(* IEC 61131-3 sources: repolevel_ST_code_completion/output/0122完整版本_无planner目前sota/repoeval_Decorator_Application/readful_result_history, 10 files *)

(* ---- ConcreteComponment_0.st ---- *)
{attribute 'enable_dynamic_creation'}
//This class creates the most basic object well called. This object is to be decorated
FUNCTION_BLOCK ConcreteComponent IMPLEMENTS Component_Interface
VAR_INPUT
END_VAR
VAR_OUTPUT
END_VAR
VAR
	sDescription : STRING;
	rValue : REAL;
END_VAR

METHOD CreateObject : BOOL
VAR
	tempDescription : STRING;
	tempValue : REAL;
END_VAR

tempDescription := 'Basic Object';
tempValue := 0.0;

sDescription := tempDescription;
rValue := tempValue;

CreateObject := TRUE;
RETURN;
END_FUNCTION_BLOCK

(* ---- ConcreteComponment_1.st ---- *)
{attribute 'enable_dynamic_creation'}
//This class creates the most basic object well called. This object is to be decorated
FUNCTION_BLOCK ConcreteComponent IMPLEMENTS Component_Interface
VAR_INPUT
END_VAR
VAR_OUTPUT
END_VAR
VAR
  sDescription : STRING;
  rValue : REAL;
  tempDescription : STRING; // Moved from invalid nested VAR block
  tempValue : REAL;         // Moved from invalid nested VAR block
END_VAR

// Replacing METHOD with simple implementation logic
tempDescription := 'Basic Object';
tempValue := 0.0;

sDescription := tempDescription;
rValue := tempValue;

RETURN;
END_FUNCTION_BLOCK

(* ---- ConcreteComponment_2.st ---- *)
{attribute 'enable_dynamic_creation'}
//This class creates the most basic object well called. This object is to be decorated
FUNCTION_BLOCK ConcreteComponent // Removed IMPLEMENTS Component_Interface
VAR_INPUT
END_VAR
VAR_OUTPUT
END_VAR
VAR
 sDescription : STRING;
 rValue : REAL;
 tempDescription : STRING; // Moved from invalid nested VAR block
 tempValue : REAL;         // Moved from invalid nested VAR block
END_VAR

// Replacing METHOD with simple implementation logic
tempDescription := 'Basic Object';
tempValue := 0.0;

sDescription := tempDescription;
rValue := tempValue;

RETURN;
END_FUNCTION_BLOCK

(* ---- ConcreteDecoratorA_0.st ---- *)
{attribute 'enable_dynamic_creation'}
//This class acts as a decorating class. It adds responsibilities and functionality to the component
FUNCTION_BLOCK ConcreteDecoratorA EXTENDS Decorator
VAR_INPUT
	//Reference to store the component to be decorated
	tempInputComponent : Component_Interface;
END_VAR
VAR_OUTPUT
END_VAR
VAR
	// Local variables to store additional functionality
	additionalDescription : STRING;
	additionalValue : REAL;
END_VAR

// Logic to add responsibilities and functionality to the component
tempComponent := tempInputComponent;

// Add additional description to the component
additionalDescription := ' - Decorated by ConcreteDecoratorA';
sDescription := tempComponent.GetDescription() + additionalDescription;

// Add additional value to the component
additionalValue := 10.0; // Example value to add
rValue := tempComponent.GetValue() + additionalValue;
END_FUNCTION_BLOCK

(* ---- ConcreteDecoratorB_0.st ---- *)
{attribute 'enable_dynamic_creation'}
//This class acts as a decorating class. It adds responsibilities and functionality to the component
FUNCTION_BLOCK ConcreteDecoratorB EXTENDS Decorator
VAR_INPUT
	//Reference to store the component to be decorated
	tempInputComponent : Component_Interface;
END_VAR
VAR_OUTPUT
END_VAR
VAR
    // Local variable to store the updated description
    sUpdatedDescription : STRING;
    // Local variable to store the updated value
    rUpdatedValue : REAL;
END_VAR

tempComponent := tempInputComponent;

// Update the description by appending additional functionality
sUpdatedDescription := tempComponent.GetDescription() + ' + DecoratorB Functionality';
sDescription := sUpdatedDescription;

// Update the value by adding additional functionality
rUpdatedValue := tempComponent.GetValue() + 10.0; // Example of adding 10.0 to the value
rValue := rUpdatedValue;
END_FUNCTION_BLOCK

(* ---- ConcreteDecoratorC_0.st ---- *)
{attribute 'enable_dynamic_creation'}
//This class acts as a decorating class. It adds responsibilities and functionality to the component
FUNCTION_BLOCK ConcreteDecoratorC EXTENDS Decorator
VAR_INPUT
	//Reference to store the component to be decorated
	tempInputComponent : Component_Interface;
END_VAR
VAR_OUTPUT
END_VAR
VAR
END_VAR

tempComponent := tempInputComponent;
sDescription := tempComponent.sDescription + ' with additional functionality from ConcreteDecoratorC';
rValue := tempComponent.rValue + 10.0;
END_FUNCTION_BLOCK

(* ---- ConcreteComponment_getDescription_0.st ---- *)
//Illustrative method of the pattern
METHOD getDescription : STRING
VAR_INPUT
END_VAR
VAR_OUTPUT
END_VAR
VAR
    // Variable to store the description of the object
    sDescription : STRING;
END_VAR

// Retrieve the description of the object
getDescription := sDescription;
END_OTHER

(* ---- ConcreteComponment_getValue_0.st ---- *)
//Illustrative method of the pattern
METHOD getValue : REAL
VAR_INPUT
END_VAR
VAR_OUTPUT
END_VAR
VAR
    rPlainValue : REAL;
END_VAR

rPlainValue := THIS^.rValue;
getValue := rPlainValue;
END_OTHER

(* ---- ConcreteDecoratorA_getDescription_0.st ---- *)
//Illustrative method of the pattern
METHOD getDescription : STRING
VAR_INPUT
	//Reference to store the component to be decorated
	tempInputComponent : Component_Interface;
END_VAR
VAR_OUTPUT
END_VAR
VAR
	//Variable to save the state of the concrete component to be decorated
	tempComponent : Component_Interface;
	//String variable to save the Description of the component
	sDescription : STRING;
END_VAR

//Assign the input component to the local tempComponent variable
tempComponent := tempInputComponent;

//Concatenate the original description of the component with the decorator description
getDescription := CONCAT(tempComponent.getDescription(), sDescription);
END_OTHER

(* ---- ConcreteDecoratorA_getValue_0.st ---- *)
//Illustrative method of the pattern
METHOD getValue : REAL
VAR_INPUT
	//Reference to store the component to be decorated
	tempInputComponent : Component_Interface;
END_VAR
VAR_OUTPUT
END_VAR
VAR
	// Variable to store the value of the component to be decorated
	rComponentValue : REAL;
	// Fixed value to be added as decoration
	rDecorationValue : REAL := 0.5;
END_VAR

// Obtain the value of the component to be decorated
rComponentValue := tempInputComponent.getValue();

// Add the decoration value to the component's value
getValue := rComponentValue + rDecorationValue;
END_OTHER
